{region '#Template'}
	{attribute 'Category' := 'Universal'}
	{attribute 'Version' := '0.0.1.0'}
	{attribute 'Tags' := 'Universal, Damper, Aggregate'}
	{attribute 'Description' := '2 Punkt Klappe mit Endlagenschalter	// 2 point damper with limit switch'}
{endregion}
FUNCTION_BLOCK FB_BA_Dmp2P EXTENDS FB_BA_AggregateB
VAR_OUTPUT
	bCmd					: BOOL;
	bSwiOpn					: BOOL;
	bSwiCls					: BOOL;
	bDstb					: BOOL;
END_VAR
VAR_INPUT CONSTANT PERSISTENT
	{attribute 'parameterCategory' := 'Behaviour'}
	{attribute 'parameterUnit':= 's'}
	nInterruptionDelay : UDINT := 1;
END_VAR
VAR_INPUT CONSTANT
	SwiOpn					: FB_BA_BI_IO;
	SwiCls					: FB_BA_BI_IO;
	Cmd						: FB_BA_BO_IO;
	MonitOpen				: FB_BA_FdbBinary;
	MonitClose				: FB_BA_FdbBinary;
END_VAR	
VAR	
END_VAR

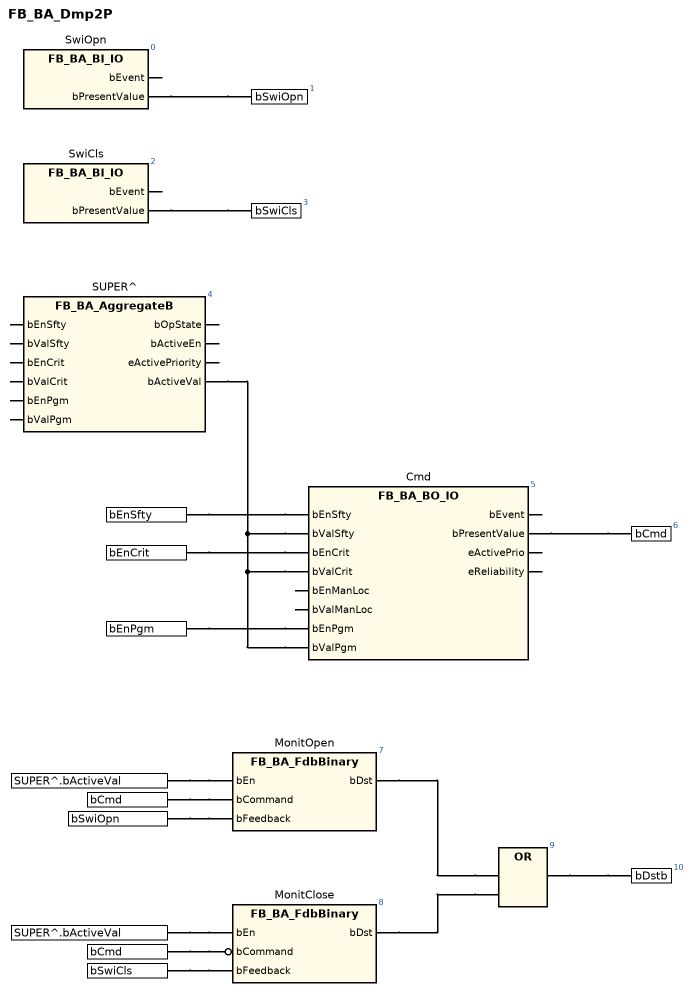
SwiOpn(); // FB_BA_BI_IO
bSwiOpn := SwiOpn.bPresentValue;
SwiCls(); // FB_BA_BI_IO
bSwiCls := SwiCls.bPresentValue;
SUPER^(); // FB_BA_AggregateB
Cmd(
    bEnSfty := bEnSfty,
    bValSfty := SUPER^.bActiveVal,
    bEnCrit := bEnCrit,
    bValCrit := SUPER^.bActiveVal,
    bEnPgm := bEnPgm,
    bValPgm := SUPER^.bActiveVal); // FB_BA_BO_IO
bCmd := Cmd.bPresentValue;
MonitOpen(bEn := SUPER^.bActiveVal, bCommand := bCmd, bFeedback := bSwiOpn); // FB_BA_FdbBinary
MonitClose(bEn := SUPER^.bActiveVal, bCommand := NOT bCmd, bFeedback := bSwiCls); // FB_BA_FdbBinary
bDstb := MonitOpen.bDst OR MonitClose.bDst;

METHOD FB_init : BOOL
VAR_INPUT
	bInitRetains : BOOL; // if TRUE, the retain variables are initialized (warm start / cold start)
	bInCopyCode : BOOL;  // if TRUE, the instance afterwards gets moved into the copy code (online change)
END_VAR
SwiOpn.iParent							:= THIS^;
SwiOpn.iLabel							:= LblUniFieldDevice.Dmp_SwiOpn;	
SwiOpn.sObjectName						:= '{Idx=01}';	
SwiOpn.sDeviceType						:= '';
SwiOpn.bEnOutOfService					:= FALSE;
SwiOpn.ePolarity						:= E_BA_Polarity.eReverse;
SwiOpn.sActiveText 						:= Texts.txtReached;
SwiOpn.sInactiveText 					:= Texts.txtNotReached;
SwiOpn.nStateChangeCount				:= 0;
SwiOpn.nActiveTimeElapsed				:= 0;
SwiOpn.nEventClassID					:= EventClasses.NotificationSimple;
SwiOpn.stTimeDelay.nToNormal			:= BA2_Param.nDefTimeDelay_ToNormal;
SwiOpn.stTimeDelay.nToAbnormal			:= BA2_Param.nDefTimeDelay_ToAbnormal;
SwiOpn.bAlarmValue						:= TRUE;
SwiOpn.bAcknowledgeRm					:= FALSE;	
SwiOpn.aEventTransitionText[1]			:= Texts.txtNone;
SwiOpn.aEventTransitionText[2]			:= Texts.txtNone;
SwiOpn.aEventTransitionText[3]			:= Texts.txtNone;
SwiOpn.bEventDetectionEnable			:= FALSE;
SwiOpn.eEnPlantLock						:= E_BA_LockPriority.eNoLock;	

SwiCls.iParent							:= THIS^;
SwiCls.iLabel							:= LblUniFieldDevice.Dmp_SwiCls;	
SwiCls.sObjectName						:= '{Idx=01}';	
SwiCls.sDeviceType						:= '';
SwiCls.bEnOutOfService					:= FALSE;
SwiCls.ePolarity						:= E_BA_Polarity.eReverse;
SwiCls.sActiveText 						:= Texts.txtReached;
SwiCls.sInactiveText 					:= Texts.txtNotReached;
SwiCls.nStateChangeCount				:= 0;
SwiCls.nActiveTimeElapsed				:= 0;
SwiCls.nEventClassID					:= EventClasses.NotificationSimple;
SwiCls.stTimeDelay.nToNormal			:= BA2_Param.nDefTimeDelay_ToNormal;
SwiCls.stTimeDelay.nToAbnormal			:= BA2_Param.nDefTimeDelay_ToAbnormal;
SwiCls.bAlarmValue						:= TRUE;
SwiCls.bAcknowledgeRm					:= FALSE;		
SwiCls.aEventTransitionText[1]			:= Texts.txtNone;
SwiCls.aEventTransitionText[2]			:= Texts.txtNone;
SwiCls.aEventTransitionText[3]			:= Texts.txtNone;
SwiCls.bEventDetectionEnable			:= FALSE;
SwiCls.eEnPlantLock						:= E_BA_LockPriority.eNoLock;

Cmd.iParent							:= THIS^;
Cmd.iLabel							:= LblUniFieldDevice.Dmp_Cmd;			
Cmd.sObjectName						:= '{Idx=01}';	
Cmd.sDeviceType						:= '';
Cmd.ePolarity						:= E_BA_Polarity.eNormal;
Cmd.eFeedbackPolarity				:= E_BA_Polarity.eNormal;
Cmd.eOverriddenPolarity				:= E_BA_Polarity.eReverse;
Cmd.sActiveText 					:= Texts.txtOn;
Cmd.sInactiveText 					:= Texts.txtOff;
Cmd.nStateChangeCount				:= 0;
Cmd.nActiveTimeElapsed				:= 0;
Cmd.nMinimumOnTime					:= 0;
Cmd.nMinimumOffTime					:= 0;
Cmd.bEnManualRm						:= FALSE;	//	Priority  8	
Cmd.bValManualRm					:= FALSE;	//	Priority  8
Cmd.bDefaultValue					:= FALSE;
Cmd.nEventClassID					:= EventClasses.DisturbanceExtended;
Cmd.stTimeDelay.nToNormal			:= BA2_Param.nDefTimeDelay_ToNormal;
Cmd.stTimeDelay.nToAbnormal			:= BA2_Param.nDefTimeDelay_ToAbnormal;
Cmd.bAcknowledgeRm					:= FALSE;		
Cmd.aEventTransitionText[1]			:= Texts.txtDisturb;
Cmd.aEventTransitionText[2]			:= Texts.txtNone;
Cmd.aEventTransitionText[3]			:= Texts.txtNormal;
Cmd.bEventDetectionEnable			:= FALSE;
Cmd.eEnPlantLock					:= E_BA_LockPriority.eNoLock;	

MonitOpen.iParent					:= THIS^;
MonitOpen.iLabel					:= LblUniFieldDevice.Dmp_Monit;	
MonitOpen.sObjectName				:= '{Idx=01}';
MonitOpen.eDPADMode					:= E_BA_DPADMode.eIncludeDescription;
MonitOpen.DelayFeedback.fValueRm	:= 180.0;

MonitClose.iParent						:= THIS^;
MonitClose.iLabel						:= LblUniFieldDevice.Dmp_Monit;	
MonitClose.sObjectName					:= '{Idx=02}';
MonitClose.eDPADMode					:= E_BA_DPADMode.eIncludeDescription;
MonitClose.DelayFeedback.fValueRm		:= 180.0;
MonitClose.DelayFeedback.sObjectName	:= '{Idx=02}';								 	 
MonitClose.Dst.sObjectName				:= '{Idx=02}';
END_METHOD

END_FUNCTION_BLOCK

(* stored: Version 1.1.0.1, ProductVersion 3.1.4024.6
   POU FB_BA_Dmp2P: Id {6fdd1ee7-14fa-421c-9872-6ba8ac973857}, SpecialFunc None
   Method FB_init: Id {e6bcaade-5b65-465e-ab86-bc6abfdd6bfa} *)
